FUNCTION GetStringSizeForS7Comm : WORD
VAR_INPUT
	stringVariable : ANY_STRING;
END_VAR

IF stringVariable.diSize < 255 THEN
	GetStringSizeForS7Comm := TO_WORD(stringVariable.diSize);
ELSE
	GetStringSizeForS7Comm := TO_WORD(stringVariable.diSize - 1);
END_IF

END_FUNCTION

(* stored: Version 1.1.0.1
   POU GetStringSizeForS7Comm: Id {69d47f42-19ea-4929-b7cd-0c97bf3a8986}, SpecialFunc None *)
